Staubli VAL3: show_check.pgx

program show_check(string x_sString_show)
begin
  userPage(sScreen_ppShelf)
  title(sScreen_ppShelf,x_sString_show)
  gotoxy(sScreen_ppShelf,0,0)
  putln(sScreen_ppShelf,"Press any key")
  //anykey
  get(sScreen_ppShelf)
  //cls(sScreen_ppShelf)
end
